RoboDK station: Assistive_UR5e _Police.rdk

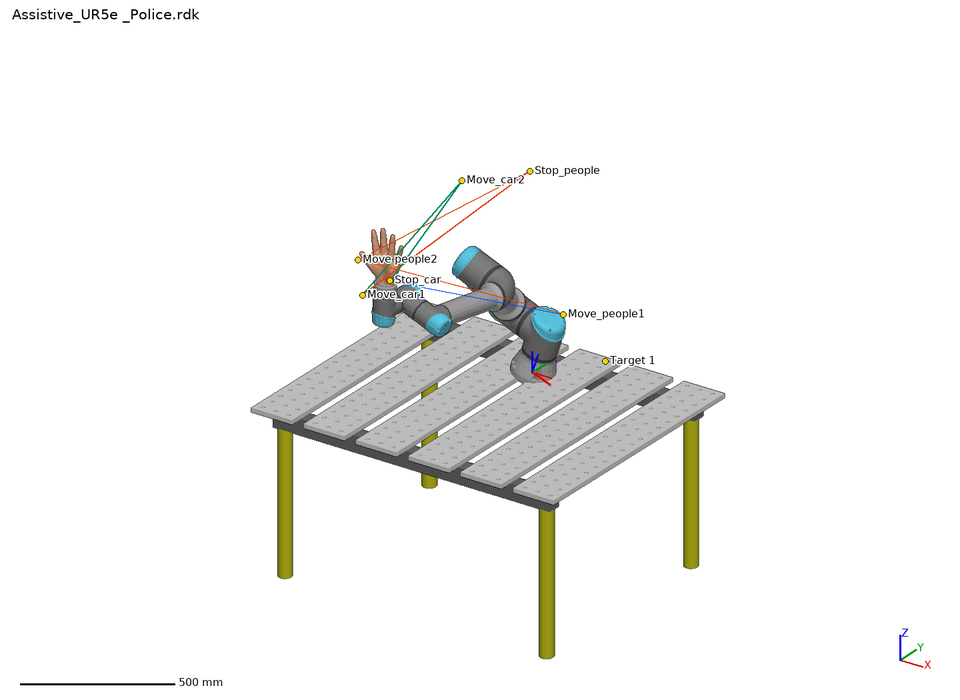
[picture v0: the station drawn from its stored meshes, robots at their saved joint values, targets as dots, program paths as lines]
Station Assistive_UR5e_SW (saved by RoboDK 5.9.2). Poses are relative to the parent item; angles as X-Y-Z fixed-axis rotations.
  - frame UR5e Base at (0, 0, 0) mm, rotated rx 0 ry 18.02 rz 0 deg
    - robot UR5e: 6 axes, payload 5 kg, reach 850 mm, repeatability 0.03 mm, weight 18.4 kg
        modified DH rows (alpha deg, a mm, theta deg, d mm): 0, 0, 0, 162.5; 90, 0, 180, 0; 0, 425, 0, 0; 0, 392.25, 0, 133.3; -90, 0, 0, 99.7; 90, 0, 180, 99.6
        joint limits [-360, -360, -360, -360, -360, -360] to [360, 360, 360, 360, 360, 360]; home [0, -90, -90, 0, 90, 0]; saved at [-94.892, -136.23, -37.635, 262.633, -75.894, 95.045]
      - tool Hand, TCP at (-17.69, -29.52, 18.63) mm, rotated rx -3.86 ry 0 rz 0 deg, size 54.8 x 155.9 x 193.5 mm, geometry from Hand.stl
    - target Target 1 (Cartesian target) at (381.17, -300.71, 440.46) mm, rotated rx 89.87 ry -18.23 rz 0.1 deg; joints [-2.034, -199.614, 94.969, 107.276, -2.134, -2.532] of UR5e
    - target Target 2 (Cartesian target) at (381.84, -300, 440.68) mm, rotated rx 90 ry -18.13 rz 0 deg; joints [-1.95, -110.285, -94.019, -155.696, -1.95, 0] of UR5e
  - frame World at (0, 0, 0) mm
    - object Table at (0, 0, 0) mm, size 1193.8 x 965.2 x 609.6 mm, geometry from welding_table.sld
    - target Stop_car (Cartesian target) at (0, -800, 650) mm, rotated rx 0 ry 0 rz 90 deg; joints [-94.892, -172.301, 37.635, 223.433, -75.894, 95.045] of UR5e
    - target Move_people1 (joint target) at (424.37, -430, 500) mm, rotated rx 90 ry 0 rz 0 deg; joints [-31.749, -180.278, 98.382, 255.171, -326.875, 203.694] of UR5e
    - target Move people2 (joint target) at (-350, -480, 500) mm, rotated rx 90 ry 0 rz 0 deg; joints [-130.206, -206.624, 85.816, 295.922, -228.702, 194.826] of UR5e
    - target Stop_people (joint target) at (200, -300, 900) mm, rotated rx 0 ry 0 rz 90 deg; joints [-80.493, -140.195, 74.619, 157.962, -76.04, 80.201] of UR5e
    - target Move_car1 (joint target) at (-130, -770, 550) mm, rotated rx -0.7 ry 38.16 rz -92.02 deg; joints [-97.31, -129.567, -54.282, 231.892, -76.402, 285.722] of UR5e
    - target Move_car2 (Cartesian target) at (-113.18, -233.59, 751.95) mm, rotated rx -0.55 ry 6.04 rz -91.65 deg; joints [-116.637, -69.289, -103.975, 247.804, -73.758, 297.981] of UR5e
  - program Stop (4 instructions, listed below)
  - program Move_people (6 instructions, listed below)
  - program Move_car (5 instructions, listed below)
  - program Main_program (3 instructions, listed below)
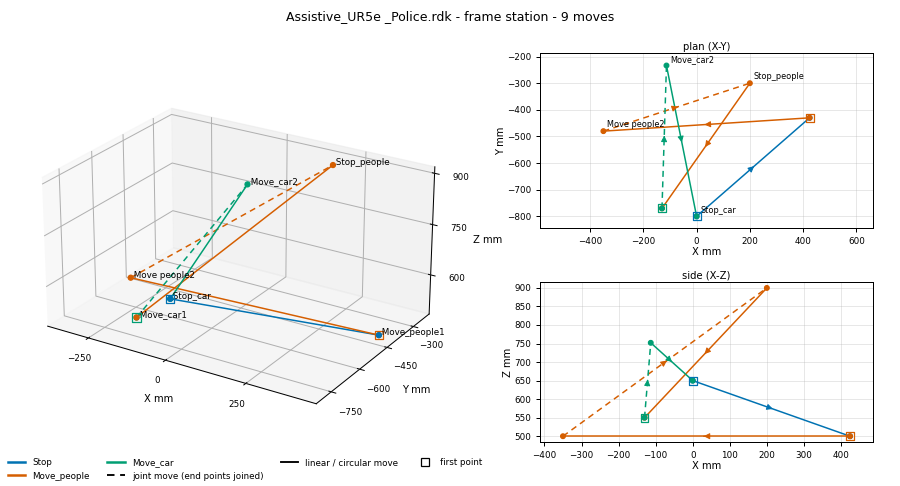
[picture p0: tool path of Assistive_UR5e _Police.rdk in frame station, 9 of 9 moves have a stored position in this frame; points joined in program order, loops and branches not executed]

--- program Stop (robot UR5e) ---
  Set Ref.: World
  Set Tool: Hand
  MoveJ (Stop_car)
  MoveL (Move_people1)

--- program Move_people (robot UR5e) ---
  Set Ref.: World
  Set Tool: Hand
  MoveJ (Move_people1)
  MoveL (Move people2)
  MoveJ (Stop_people)
  MoveL (Move_car1)

--- program Move_car (robot UR5e) ---
  Set Ref.: World
  Set Tool: Hand
  MoveJ (Move_car1)
  MoveJ (Move_car3) -> target Move_car2
  MoveL (Stop_car)

--- program Main_program (robot UR5e) ---
  Call Stop
  Call Move_people
  Call Move_car
